PROGRAM EspNodeController
VAR
	EspFactory			: EspNodeFactory;
	List				: List(EspFactory);
	Node				: ITF_Node;
	NodePtr				: POINTER TO EspHost;
	EspDevice			: ITF_EspHost;
	ListIndex			: UINT;
	CreateEspDevice		: BOOL;
	DestroyEspDevice	: BOOL;
	GetEspDevice		: BOOL;
END_VAR

IF CreateEspDevice THEN

	IF List.CreateNode() THEN
		
		CreateEspDevice := FALSE;
		
	END_IF

END_IF

IF DestroyEspDevice THEN

	IF List.DestroyNode(ListIndex) THEN
		
		DestroyEspDevice := FALSE;
		
	END_IF

END_IF

IF GetEspDevice THEN

	Node := List.GetNode(ListIndex);
	
	NodePtr := Node.GetMyPointer();
	
	EspDevice := NodePtr^;
	
	IF EspDevice <> 0 THEN
		
		GetEspDevice := FALSE;
		
	END_IF

END_IF

END_PROGRAM

(* stored: Version 1.1.0.1
   POU EspNodeController: Id {c6bd84ac-1a70-48cb-b8d1-05da0a65a282}, SpecialFunc None *)
